PROGRAM MAIN
VAR
END_VAR

Alias();
Heartbeat();
Permissives();
Trips();
Alarms();
Sequence();

END_PROGRAM

(* stored: Version 1.1.0.1, ProductVersion 3.1.4024.11
   POU MAIN: Id {d4510c44-5a58-4477-924a-86d697b0947a}, SpecialFunc None *)
